Universal Robots PolyScope program: T03_conditional_teleop.urp

Program T03_conditional_teleop (installation=default directory=/programs createdIn=5.9.1.1031110 lastSavedIn=5.9.1.1031110 robotSerialNumber=20195501059)
Calibrated DH parameters: a=[0.000146, -0.418764, -0.053981, 0.000058, -0.000023, 0]; d=[0.162545, 37.319448, -206.067439, 168.881546, 0.09955, 0.099464]; alpha=[1.57004, -0.001979, 0.002304, 1.570607, -1.57066, 0]; deltaTheta=[0, -0.174616, -1.258233, 1.432844, -0.000001, 0]
BeforeStart
  URCap Gripper Activate (Robotiq_Grippers, Robotiq Inc.) dataModel(ResetAndActivateKey=false)
  start_p := get_actual_tcp_pose()
  MoveJ speed 60 deg/s, acceleration 80 deg/s^2 (useActiveTCP=true) feature=Base
    Waypoint Waypoint (Variable): variable=start_p
Robot Program (runOnlyOnce=false)
  MoveL speed 250 mm/s, acceleration 1200 mm/s^2 (useActiveTCP=true) feature=Base
    Waypoint approach_p: TCP in base x=149.271 y=-546.431 z=71.633 mm, rx=2.2516 ry=2.1906 rz=-0.0002 rad; joints [91.615, -72.502, 107.097, -124.599, 270.032, 93.216] deg; TCP offset x=0 y=0 z=174 mm, rx=0 ry=0 rz=0 rad
    URCap Gripper (Robotiq_Grippers, Robotiq Inc.) dataModel(position=55.0, force=0.0, speed=100.0, positionInDouble=55.0, forceInDouble=0.0, speedInDouble=100.0, slaveIds=[9], blocking=true)
    Waypoint grasp_p: TCP in base x=149.291 y=-546.451 z=22.049 mm, rx=2.2516 ry=2.1906 rz=-0.0002 rad; joints [91.613, -68.141, 109.925, -131.789, 270.037, 93.222] deg
    URCap Gripper (Robotiq_Grippers, Robotiq Inc.) dataModel(position=100.0, force=0.0, speed=100.0, positionInDouble=100.0, forceInDouble=0.0, speedInDouble=100.0, slaveIds=[9], blocking=true)
    URCap Grip Check (Robotiq_Grippers, Robotiq Inc.) dataModel(ObjectDetectedKey=true, DimensionValidationKey=false, DimensionKey=100.0, DimensionDimensionPositiveGapKey=5.0, DimensionNegativeGapKey=5.0, GripperIdKey=1, ModelDefinedKey=true); state(isChildrenLocked=true)
      URCap If (Robotiq_Grippers, Robotiq Inc.)
        URCap Gripper (Robotiq_Grippers, Robotiq Inc.) dataModel(position=55.0, force=0.0, speed=100.0, positionInDouble=55.0, forceInDouble=0.0, speedInDouble=100.0, slaveIds=[9], blocking=true)
        MoveL speed 250 mm/s, acceleration 1200 mm/s^2 (useActiveTCP=true) feature=Base
          Waypoint approach_p: TCP in base x=149.271 y=-546.431 z=71.633 mm, rx=2.2516 ry=2.1906 rz=-0.0002 rad; joints [91.615, -72.502, 107.097, -124.599, 270.032, 93.216] deg
      URCap Else (Robotiq_Grippers, Robotiq Inc.)
        URCap Olis Teleop (Olis Teleop, Olis Robotics) dataModel(OperatorMessage=Please troubleshoot- missing part)
        MoveL speed 250 mm/s, acceleration 1200 mm/s^2 (useActiveTCP=true) feature=Base
          Waypoint approach_p: TCP in base x=149.271 y=-546.431 z=71.633 mm, rx=2.2516 ry=2.1906 rz=-0.0002 rad; joints [91.615, -72.502, 107.097, -124.599, 270.032, 93.216] deg
